// TIA Portal V19 export
FUNCTION "Output_Peripherie" : Void   // FC1011, LAD
{ S7_Optimized_Access := 'TRUE' }
// stored: AutoNumber false, SetENOAutomatically true
BEGIN

REGION Network 1 (SCL): Schnellauftor
   "A_RT_auf" := "Tor".Out.auf;
   "A_RT_zu" := "Tor".Out.zu;
END_REGION

REGION Network 2 (SCL): Deckel
   // CM01
   "A_Dkl_li_auf_CM01" := "Deckel_CM01".Out.links_auf;
   "A_Dkl_li_zu_CM01" := "Deckel_CM01".Out.links_zu;
   "A_Dkl_re_auf_CM01" := "Deckel_CM01".Out.rechts_auf;
   "A_Dkl_re_zu_CM01" := "Deckel_CM01".Out.rechts_zu;
   // CM02
   "A_Dkl_li_auf_CM02" := "Deckel_CM02".Out.links_auf;
   "A_Dkl_li_zu_CM02" := "Deckel_CM02".Out.links_zu;
   "A_Dkl_re_auf_CM02" := "Deckel_CM02".Out.rechts_auf;
   "A_Dkl_re_zu_CM02" := "Deckel_CM02".Out.rechts_zu;
END_REGION

REGION Network 3 (SCL): CM01
   //Filtern
   // Pumpe (FU[1])
   "A_Frg_FU_FP_HQ01" := "FP_CM01.GP01".Out.GP0x_Ein;

   "FU_In_Out".FU[1].PA.Steuerwort.FrgHalt := "FP_CM01.GP01".Out.GP0x_Ein;
   "FU_In_Out".FU[1].PA.Steuerwort.FrgStop := "FP_CM01.GP01".Out.GP0x_Ein;
   "FU_In_Out".FU[1].PA.Steuerwort.RegSp := NOT "FU_In_Out".FU[1].PA.Steuerwort.FrgHalt;
   "FU_In_Out".FU[1].PA.Speed := "FP_CM01.GP01".Out.Soll_speed;

   // IF ("FP_CM01.GP01".In."Betriebsart" = 0) AND ("Panel".FP_CM01.BA = 1) THEN
   //     "Panel".FP_CM01.BA := 0; // Filtern
   // END_IF;

   //Ventile
   "A_CM01.QM18" := "FP_CM01.GP01".Out.Ventil_Saugseite;
   "A_CM01.QM19" := "FP_CM01.GP01".Out.Spülventil_P_Eingang;
   "A_HQ01.LV01" := "FP_CM01.GP01".Out.Ventil_Entlueften;
   "A_HQ01.QM21" := "FP_CM01.GP01".Out.Ventil_Eingang_Filter;
   "A_HQ01.QM22" := "FP_CM01.GP01".Out.Spülventil_F_Eingang;
   "A_HQ01.QM23" := "FP_CM01.GP01".Out.Ventil_Ausgang_Filter;
   "A_HQ01.QM24" := "FP_CM01.GP01".Out.Spülventil_Ausgang;

   // Umwälzen
   // Pumpe (FU[2])
   "A_Frg_FU_UP_HF_CM01" := "UP_CM01.GP02".Out.GP0x_Ein;

   "FU_In_Out".FU[2].PA.Steuerwort.FrgHalt := "UP_CM01.GP02".Out.GP0x_Ein;
   "FU_In_Out".FU[2].PA.Steuerwort.FrgStop := "UP_CM01.GP02".Out.GP0x_Ein;
   "FU_In_Out".FU[2].PA.Steuerwort.RegSp := NOT "FU_In_Out".FU[2].PA.Steuerwort.FrgHalt;
   "FU_In_Out".FU[2].PA.Speed := "UP_CM01.GP02".Out.Soll_speed;

   //Ventile
   "A_CM01.QM25" := "UP_CM01.GP02".Out.Ventil_Saugseite;
   "A_CM01.QM26" := "UP_CM01.GP02".Out.Ventil_Druckseite;
   "A_CM01.QM20" := "UP_CM01.GP02".Out.Spülventil_Eingang;
   "A_CM01.QM27" := "UP_CM01.GP02".Out.Spülventil_Ausgang;
   "A_GP02.QM45":= "UP_CM01.GP02".Out.Entsorgung_UV02;
   "A_GP02.QM44" := "UP_CM01.GP02".Out.Ventil_UV02_GP01 OR "UP_CM02.GP05".Out.Ventil_UV02_GP01;
   "A_GP02.QM43" := "UP_CM01.GP02".Out.Ventil_UV02_GP02 OR "UP_CM02.GP05".Out.Ventil_UV02_GP02;
END_REGION

REGION Network 4 (SCL): CM02
   //Filtern
   // Pumpe (FU[4])
   "A_Frg_FU_FP_HQ02" := "FP_CM02.GP04".Out.GP0x_Ein;

   "FU_In_Out".FU[4].PA.Steuerwort.FrgHalt := "FP_CM02.GP04".Out.GP0x_Ein;
   "FU_In_Out".FU[4].PA.Steuerwort.FrgStop := "FP_CM02.GP04".Out.GP0x_Ein;
   "FU_In_Out".FU[4].PA.Steuerwort.RegSp := NOT "FU_In_Out".FU[4].PA.Steuerwort.FrgHalt;
   "FU_In_Out".FU[4].PA.Speed := "FP_CM02.GP04".Out.Soll_speed;

   // IF ("FP_CM02.GP04".In."Betriebsart" = 0) AND ("Panel".FP_CM02.BA = 1) THEN
   //     "Panel".FP_CM02.BA := 0; // Filtern
   // END_IF;

   //Ventile
   "A_CM02.QM55" := "FP_CM02.GP04".Out.Ventil_Saugseite;
   "A_CM02.QM56" := "FP_CM02.GP04".Out.Spülventil_P_Eingang;
   "A_HQ02.LV02" := "FP_CM02.GP04".Out.Ventil_Entlueften;
   "A_HQ02.QM59" := "FP_CM02.GP04".Out.Ventil_Eingang_Filter;
   "A_HQ02.QM58" := "FP_CM02.GP04".Out.Spülventil_F_Eingang;
   "A_HQ02.QM60" := "FP_CM02.GP04".Out.Ventil_Ausgang_Filter;
   "A_HQ02.QM61" := "FP_CM02.GP04".Out.Spülventil_Ausgang;

   // Umwälzen
   // Pumpe (FU[5])
   "A_Frg_FU_UP_HF_CM02" := "UP_CM02.GP05".Out.GP0x_Ein;

   "FU_In_Out".FU[5].PA.Steuerwort.FrgHalt := "UP_CM02.GP05".Out.GP0x_Ein;
   "FU_In_Out".FU[5].PA.Steuerwort.FrgStop := "UP_CM02.GP05".Out.GP0x_Ein;
   "FU_In_Out".FU[5].PA.Steuerwort.RegSp := NOT "FU_In_Out".FU[5].PA.Steuerwort.FrgHalt;
   "FU_In_Out".FU[5].PA.Speed := "UP_CM02.GP05".Out.Soll_speed;

   //Ventile
   "A_CM02.QM62" := "UP_CM02.GP05".Out.Ventil_Saugseite;
   "A_CM02.QM63" := "UP_CM02.GP05".Out.Ventil_Druckseite;
   "A_CM02.QM57" := "UP_CM02.GP05".Out.Spülventil_Eingang;
   "A_CM02.QM64" := "UP_CM02.GP05".Out.Spülventil_Ausgang;
   "A_GP02.QM46" := "UP_CM02.GP05".Out.Entsorgung_UV02;
END_REGION

REGION Network 5 (SCL): CM03
   // Pumpe (FU[3])
   "A_Frg_FU_UP_H2O_CM03" := "UP_CM03.GP03".Out.GP0x_Ein;

   "FU_In_Out".FU[3].PA.Steuerwort.FrgHalt := "UP_CM03.GP03".Out.GP0x_Ein;
   "FU_In_Out".FU[3].PA.Steuerwort.FrgStop := "UP_CM03.GP03".Out.GP0x_Ein;
   "FU_In_Out".FU[3].PA.Steuerwort.RegSp := NOT "FU_In_Out".FU[3].PA.Steuerwort.FrgHalt;
   "FU_In_Out".FU[3].PA.Speed := "UP_CM03.GP03".Out.Soll_speed;

   // Ventile
   "A_CM03.QM33" := "UP_CM03.GP03".Out.Ventil_Saugseite;
   "A_CM03.QM34" := "UP_CM03.GP03".Out.Ventil_Druckseite;
   "A_CM03.QM36" := "UP_CM03.GP03".Out.Spülventil;
   "A_CM03.QM37" := "UP_CM03.GP03".Out.Ventil_CM05;
END_REGION

REGION Network 6 (SCL): CM04
   // Pumpe (FU[6])
   "A_Frg_FU_UP_H2O_CM04" := "UP_CM04.GP06".Out.GP0x_Ein;

   "FU_In_Out".FU[6].PA.Steuerwort.FrgHalt := "UP_CM04.GP06".Out.GP0x_Ein;
   "FU_In_Out".FU[6].PA.Steuerwort.FrgStop := "UP_CM04.GP06".Out.GP0x_Ein;
   "FU_In_Out".FU[6].PA.Steuerwort.RegSp := NOT "FU_In_Out".FU[6].PA.Steuerwort.FrgHalt;
   "FU_In_Out".FU[6].PA.Speed := "UP_CM04.GP06".Out.Soll_speed;

   // Ventile
   "A_CM04.QM72" := "UP_CM04.GP06".Out.Ventil_Saugseite;
   "A_CM04.QM73" := "UP_CM04.GP06".Out.Ventil_Druckseite;
   "A_CM04.QM75" := "UP_CM04.GP06".Out.Spülventil;
   "A_CM04.QM76" := "UP_CM04.GP06".Out.Ventil_CM05;
END_REGION

REGION Network 7 (SCL): CM05
   // Pumpe
   "A_Pu_Entl_CM05" := "Pu_CM05.GP11_DB".Out.GP11_Ein;
   // Ventile
   "A_CM05.QM61" := "Pu_CM05.GP11_DB".Out.QM61;
   "A_CM05.QM62" := "Pu_CM05.GP11_DB".Out.QM62;
   "A_CM05.QM63" := "Pu_CM05.GP11_DB".Out.QM63;
   "A_CM05.QM64" := "Pu_CM05.GP11_DB".Out.QM64;
END_REGION

REGION Network 8 (SCL): CL0x
   // CL01
   // Pumpe
   "A_CL01.GP08" := "Pu_CL01.GP08".Out.GP0x_Ein;
   // Spülventil
   "A_CL01.QM51" := "Pu_CL01.GP08".Out.Spülventil;

   // CL02
   // Pumpe
   "A_CL02.GP09" := "Pu_CL02.GP09".Out.GP0x_Ein;
   // Spülventil
   "A_CL02.QM52" := "Pu_CL02.GP09".Out.Spülventil;
END_REGION

REGION Network 9 (SCL): GP01
   // Versorgung
   // Pumpe
   "A_GP01.GP13" := "Pu_GP01.GP13".Out.GP0x_Ein;
   // Ventile
   "A_GP01.QM14" := "Pu_GP01.GP13".Out.Ventil_Entsorgung;
   "A_GP01.QM15" := "Pu_GP01.GP13".Out.Ventil_Saugseite;
   "A_GP01.QM16" := "Pu_GP01.GP13".Out.Spülventil_Eingang;
   "A_GP01.QM17" := "Pu_GP01.GP13".Out.Spülventil_Ausgang;
   "A_GP01.QM18" := "Pu_GP01.GP13".Out.Ventil_Druckseite;
   "A_GP01.QM22" := "Pu_GP01.GP13".Out.Versorgung_UV01;

   "A_GP01.QM19" := "Pu_GP01.GP13".Out.UV01_CM02 OR "Pu_GP02.GP10".Out.UV01_CM02;
   "A_GP01.QM20" := "Pu_GP01.GP13".Out.UV01_CM01 OR "Pu_GP02.GP10".Out.UV01_CM01;

   // Entleeren Sumpf
   // Pumpe
   "A_GP01.GP12" := "Pu_GP01.GP12".Out.GP0x_Ein AND "DB_PNOZ_IN_Out".In.Tuer_zu_Seite_GP01 AND "DB_PNOZ_IN_Out".In.Tuer_zu_vorn_GP01;
   // Spülventil
   "A_GP01.QM23" := "Pu_GP01.GP12".Out.Spülventil AND "DB_PNOZ_IN_Out".In.Tuer_zu_Seite_GP01 AND "DB_PNOZ_IN_Out".In.Tuer_zu_vorn_GP01;
   // IBC
   "A_IBC_Vers" := "E_S_IBC_GP01.BG21";
END_REGION

REGION Network 10 (SCL): GP02
   // Versorgung
   // Pumpe
   "A_GP02.GP10" := "Pu_GP02.GP10".Out.GP0x_Ein;
   // Ventile
   "A_GP02.QM41" := "Pu_GP02.GP10".Out.Ventil_Entsorgung;
   "A_GP02.QM38" := "Pu_GP02.GP10".Out.Ventil_Saugseite;
   "A_GP02.QM39" := "Pu_GP02.GP10".Out.Spülventil_Eingang;
   "A_GP02.QM42" := "Pu_GP02.GP10".Out.Spülventil_Ausgang;
   "A_GP02.QM40" := "Pu_GP02.GP10".Out.Ventil_Druckseite;
   "A_GP01.QM21" := "Pu_GP02.GP10".Out.Versorgung_UV01;

   // Entleeren Sumpf
   // Pumpe
   "A_GP02.GP07" := "Pu_GP02.GP07".Out.GP0x_Ein AND "DB_PNOZ_IN_Out".In.Tuer_zu_vorn_GP02;
   // Spülventil
   "A_GP02.QM37" := "Pu_GP02.GP07".Out.Spülventil AND "DB_PNOZ_IN_Out".In.Tuer_zu_vorn_GP02;
   // IBC
   "A_IBC_Ents" := "E_S_IBC_GP02.BG22";
END_REGION
END_FUNCTION
